FUNCTION_BLOCK FB_NovRamToFileRingBuffer
VAR_INPUT
	udiNovRamIndex:UDINT;
	dataType:DINT;
END_VAR
VAR_OUTPUT
	//readData:ARRAY [0..GVL.arrArrayLength[E_DB_StructureType.AlarmHistory]-1] OF ST_AlarmInfo_DB_save;
END_VAR
VAR
END_VAR
VAR_IN_OUT
	NovRamData:ST_NovRam;
END_VAR

IF dataType = E_DB_StructureType.AlarmHistory THEN
	M_AlarmHistory(udiNovRamIndex:=udiNovRamIndex);
ELSIF dataType = E_DB_StructureType.ProductionHistory THEN
	M_ProductionHistory(udiNovRamIndex:=udiNovRamIndex);
ELSIF dataType = E_DB_StructureType.ProductionReport THEN
	M_ProductionReport(udiNovRamIndex:=udiNovRamIndex);
ELSIF dataType = E_DB_StructureType.ProductionSummary THEN
	M_ProductionSummary(udiNovRamIndex:=udiNovRamIndex);
ELSIF dataType = E_DB_StructureType.SoDuration THEN
	M_SoDuration(udiNovRamIndex:=udiNovRamIndex);
ELSIF dataType = E_DB_StructureType.StopCount THEN
	M_StopCount(udiNovRamIndex:=udiNovRamIndex);
ELSIF dataType = E_DB_StructureType.RegularCheckResults THEN
	M_RegularCheckResults(udiNovRamIndex:=udiNovRamIndex);
END_IF

METHOD M_AlarmHistory : BOOL
VAR_INPUT
	udiNovRamIndex:UDINT;
END_VAR
VAR_OUTPUT
	
END_VAR
VAR_INST
	WriteData:ARRAY[0..GVL.arrArrayLength[E_DB_StructureType.AlarmHistory]-1] OF ST_AlarmInfo_DB_save;//small
	iStep:INT;
	i:UDINT;
	fbFileRingBuffer: FB_FileRingBuffer := ( sNetId     := '',
                                             sPathName  := '',
                                             ePath      := PATH_GENERIC,
                                             nID        := 1,
                                             cbBuffer   := gvl.arrFileRingBufferSize[E_DB_StructureType.AlarmHistory], //5MB(5*10^6Bytes)
                                             bOverwrite := FALSE,
                                             pWriteBuff := 0,
                                             cbWriteLen := 0,
                                             pReadBuff  := 0,
                                             cbReadLen  := 0,
                                             tTimeout   := T#1S );
	bBusy:BOOL;
	bError:BOOL;
	nErrID:UDINT;
	stHeader:ST_FileRBufferHead;
    loadData  : ARRAY[0..511] OF BYTE :=[512(0)];
    cbLoad    : UDINT;
	
	fileName:STRING(255);
	tempFileIndex:UDINT;
	eStrIndex:DINT;
	
	//1217
	TransTrig:TON;
END_VAR
//Config	
eStrIndex:=E_DB_StructureType.AlarmHistory;

fbFileRingBuffer(sPathName:=fileName
				,bBusy=>bBusy,bError=>bError,nErrID=>nErrID
				,cbReturn=>cbLoad,stHeader=>stHeader);
//1217				
TransTrig(PT:=T#10S);//10s upload one time

CASE iStep OF
	0://NovRam full detect / file full detect
		
		tempFileIndex:=NovRamData.arrFileRingBuffer_Status[eStrIndex].nowFileIndex[udiNovRamIndex];
		
		//1217
		IF NovRamData.arrNovRam_Status[eStrIndex].RowDataLocked[udiNovRamIndex] = FALSE//not full and 
		AND NovRamData.arrNovRam_Status[eStrIndex].writenIndex > 0 THEN//has been writen
			
			TransTrig(IN:=TRUE);
			
			IF TransTrig.Q //timeout
			AND NovRamData.arrFileRingBuffer_Status[eStrIndex].bFileFull[udiNovRamIndex][tempFileIndex] = FALSE THEN//File can write
				TransTrig(IN:=FALSE);
				
				//Set Row Lock
				NovRamData.arrNovRam_Status[eStrIndex].RowDataLocked[udiNovRamIndex]:=TRUE;
				
				//save writen count
				NovRamData.arrNovRam_Status[eStrIndex].writenCount := NovRamData.arrNovRam_Status[eStrIndex].writenIndex;
				
				//Reset Row and writenIndex
				NovRamData.arrNovRam_Status[eStrIndex].nowRowIndex:=(udiNovRamIndex+1)MOD GVL.NovRamBufferRatio;
				NovRamData.arrNovRam_Status[eStrIndex].writenIndex:=0;
		
				fileName:=M_GetFileName(structureType:=eStrIndex
										,udiNovRam_BufferIndex:=udiNovRamIndex
										,udiFile_Index:=NovRamData.arrFileRingBuffer_Status[eStrIndex].nowFileIndex[udiNovRamIndex]);
										
				iStep:=1;
			END_IF
			
		ELSE
			IF NovRamData.arrNovRam_Status[eStrIndex].RowDataLocked[udiNovRamIndex] //NovRam full = should work
			AND NovRamData.arrFileRingBuffer_Status[eStrIndex].bFileFull[udiNovRamIndex][tempFileIndex] = FALSE//File can write
			THEN
				//
				fileName:=M_GetFileName(structureType:=eStrIndex
										,udiNovRam_BufferIndex:=udiNovRamIndex
										,udiFile_Index:=NovRamData.arrFileRingBuffer_Status[eStrIndex].nowFileIndex[udiNovRamIndex]);
										
				iStep:=1;
			END_IF
		END_IF
		
		

	1://Open File
		
		fbFileRingBuffer.A_Open();
		
		iStep:=2;
		
	2://Wait Done/Add Data
		IF fbFileRingBuffer.bBusy=FALSE AND NOT fbFileRingBuffer.bError THEN
			
			//1217
			//FOR i:=0 TO GVL.arrArrayLength[E_DB_StructureType.AlarmHistory]-1 DO 
			FOR i:=0 TO NovRamData.arrNovRam_Status[eStrIndex].writenCount-1 DO
				WriteData[i] := NovRamData.AlarmHistory[udiNovRamIndex][i];
			END_FOR
			
			//1217
			//Add
			//fbFileRingBuffer.A_AddTail( pWriteBuff := ADR(WriteData), cbWriteLen := SIZEOF(WriteData),
			//		pReadBuff := 0, cbReadLen:=0 );
			fbFileRingBuffer.A_AddTail( pWriteBuff := ADR(WriteData), cbWriteLen := NovRamData.arrNovRam_Status[eStrIndex].writenCount * SIZEOF(ST_AlarmInfo_DB_save),
					pReadBuff := 0, cbReadLen:=0 );
					
			iStep:=3;
			
		END_IF
	3://Wait Done / Close file /(Check if file Full)
		IF fbFileRingBuffer.bBusy=FALSE THEN
						
			//Check if file full
			IF NOT fbFileRingBuffer.bError THEN
				iStep:=4;
			ELSIF fbFileRingBuffer.bError = TRUE AND nErrID=32768 THEN//full
				iStep:=11;
			END_IF
			
			//close file
			fbFileRingBuffer.A_Close();
			
		END_IF
	4://Wait Done(file still has space)
		IF fbFileRingBuffer.bBusy=FALSE AND NOT fbFileRingBuffer.bError THEN
			
			NovRamData.arrNovRam_Status[eStrIndex].RowDataLocked[udiNovRamIndex]:=FALSE;
			
			iStep:=0;
		END_IF
	11://Wait Done(file full)
		IF fbFileRingBuffer.bBusy=FALSE AND NOT fbFileRingBuffer.bError THEN
			
			//Lock now file
			//NovRamData.arrFileRingBuffer_Status.bFileFull[(gvl.FileRingBufferRatio * udiNovRamIndex) + NovRamData.arrFileRingBuffer_Status.nowFileIndex[udiNovRamIndex]]:=TRUE;
			tempFileIndex:=NovRamData.arrFileRingBuffer_Status[eStrIndex].nowFileIndex[udiNovRamIndex];
			NovRamData.arrFileRingBuffer_Status[eStrIndex].bFileFull[udiNovRamIndex][tempFileIndex]:=TRUE;
			
			//Move to next FileIndex
			NovRamData.arrFileRingBuffer_Status[eStrIndex].nowFileIndex[udiNovRamIndex]:=((NovRamData.arrFileRingBuffer_Status[eStrIndex].nowFileIndex[udiNovRamIndex]+1) MOD GVL.FileRingBufferRatio);
			
			iStep:=0;
			
		END_IF
END_CASE
END_METHOD

METHOD M_GetFileName : STRING(255)
VAR_INPUT
	structureType:DINT;
	udiNovRam_BufferIndex:UDINT;
	udiFile_Index:UDINT;
END_VAR
VAR
	tempString:STRING(255);
	tempString2:STRING(255);
	tempFileNo:UDINT;
END_VAR
IF structureType=E_DB_StructureType.AlarmHistory THEN
	tempString:=CONCAT(gvl.arrfileFolder[structureType],'AlarmHistory');
ELSIF structureType=E_DB_StructureType.ProductionHistory THEN
	tempString:=CONCAT(gvl.arrfileFolder[structureType],'ProductionHistory');
ELSIF structureType=E_DB_StructureType.ProductionReport THEN
	tempString:=CONCAT(gvl.arrfileFolder[structureType],'ProductionReport');
ELSIF structureType=E_DB_StructureType.ProductionSummary THEN
	tempString:=CONCAT(gvl.arrfileFolder[structureType],'ProductionSummary');
ELSIF structureType=E_DB_StructureType.SoDuration THEN
	tempString:=CONCAT(gvl.arrfileFolder[structureType],'SoDuration');
ELSIF structureType=E_DB_StructureType.StopCount THEN
	tempString:=CONCAT(gvl.arrfileFolder[structureType],'StopCount');
ELSIF structureType=E_DB_StructureType.RegularCheckResults THEN
	tempString:=CONCAT(gvl.arrfileFolder[structureType],'RegularCheckResults');
END_IF

tempFileNo:=(udiNovRam_BufferIndex) * GVL.FileRingBufferRatio + (udiFile_Index + 1);
tempString2:=CONCAT(tempString,UDINT_TO_STRING(tempFileNo));
M_GetFileName:=CONCAT(tempString2,'.dat');
END_METHOD

METHOD M_ProductionHistory : BOOL
VAR_INPUT
	udiNovRamIndex:UDINT;
END_VAR
VAR_INST
	WriteData:ARRAY[0..GVL.arrArrayLength[E_DB_StructureType.ProductionHistory]-1] OF ST_PHI_GroupData_DB;//small
	iStep:INT;
	i:UDINT;
	fbFileRingBuffer: FB_FileRingBuffer := ( sNetId     := '',
                                             sPathName  := '',
                                             ePath      := PATH_GENERIC,
                                             nID        := 1,
                                             cbBuffer   := gvl.arrFileRingBufferSize[E_DB_StructureType.ProductionHistory], //5MB(5*10^6Bytes)
                                             bOverwrite := FALSE,
                                             pWriteBuff := 0,
                                             cbWriteLen := 0,
                                             pReadBuff  := 0,
                                             cbReadLen  := 0,
                                             tTimeout   := T#1S );
	bBusy:BOOL;
	bError:BOOL;
	nErrID:UDINT;
	stHeader:ST_FileRBufferHead;
    loadData  : ARRAY[0..511] OF BYTE :=[512(0)];
    cbLoad    : UDINT;
	
	fileName:STRING(255);
	tempFileIndex:UDINT;
	eStrIndex:DINT;
END_VAR
//Config
eStrIndex:=E_DB_StructureType.ProductionHistory;

fbFileRingBuffer(sPathName:=fileName
				,bBusy=>bBusy,bError=>bError,nErrID=>nErrID
				,cbReturn=>cbLoad,stHeader=>stHeader);

CASE iStep OF
	0://NovRam full detect / file full detect
		
		tempFileIndex:=NovRamData.arrFileRingBuffer_Status[eStrIndex].nowFileIndex[udiNovRamIndex];
		
		IF NovRamData.arrNovRam_Status[eStrIndex].RowDataLocked[udiNovRamIndex] //NovRam full = should work
		AND NovRamData.arrFileRingBuffer_Status[eStrIndex].bFileFull[udiNovRamIndex][tempFileIndex] = FALSE//File can write
		THEN
			//
			fileName:=M_GetFileName(structureType:=eStrIndex
									,udiNovRam_BufferIndex:=udiNovRamIndex
									,udiFile_Index:=NovRamData.arrFileRingBuffer_Status[eStrIndex].nowFileIndex[udiNovRamIndex]);
									
			iStep:=1;
		END_IF

	1://Open File
		
		fbFileRingBuffer.A_Open();
		
		iStep:=2;
		
	2://Wait Done/Add Data
		IF fbFileRingBuffer.bBusy=FALSE AND NOT fbFileRingBuffer.bError THEN
			
			FOR i:=0 TO GVL.arrArrayLength[E_DB_StructureType.ProductionHistory]-1 DO 
				WriteData[i] := NovRamData.ProductionHistory[udiNovRamIndex][i];
			END_FOR
			
			//Add
			fbFileRingBuffer.A_AddTail( pWriteBuff := ADR(WriteData), cbWriteLen := SIZEOF(WriteData),
					pReadBuff := 0, cbReadLen:=0 );
			
			iStep:=3;
			
		END_IF
	3://Wait Done / Close file /(Check if file Full)
		IF fbFileRingBuffer.bBusy=FALSE THEN
						
			//Check if file full
			IF NOT fbFileRingBuffer.bError THEN
				iStep:=4;
			ELSIF fbFileRingBuffer.bError = TRUE AND nErrID=32768 THEN//full
				iStep:=11;
			END_IF
			
			//close file
			fbFileRingBuffer.A_Close();
			
		END_IF
	4://Wait Done(file still has space)
		IF fbFileRingBuffer.bBusy=FALSE AND NOT fbFileRingBuffer.bError THEN
			
			NovRamData.arrNovRam_Status[eStrIndex].RowDataLocked[udiNovRamIndex]:=FALSE;
			
			iStep:=0;
		END_IF
	11://Wait Done(file full)
		IF fbFileRingBuffer.bBusy=FALSE AND NOT fbFileRingBuffer.bError THEN
			
			//Lock now file
			//NovRamData.FileRingBuffer_Status.bFileFull[(gvl.FileRingBufferRatio * udiNovRamIndex) + NovRamData.FileRingBuffer_Status.nowFileIndex[udiNovRamIndex]]:=TRUE;
			tempFileIndex:=NovRamData.arrFileRingBuffer_Status[eStrIndex].nowFileIndex[udiNovRamIndex];
			NovRamData.arrFileRingBuffer_Status[eStrIndex].bFileFull[udiNovRamIndex][tempFileIndex]:=TRUE;
			
			//Move to next FileIndex
			NovRamData.arrFileRingBuffer_Status[eStrIndex].nowFileIndex[udiNovRamIndex]:=((NovRamData.arrFileRingBuffer_Status[eStrIndex].nowFileIndex[udiNovRamIndex]+1) MOD GVL.FileRingBufferRatio);
			
			iStep:=0;
			
		END_IF
END_CASE
END_METHOD

METHOD M_ProductionReport : BOOL
VAR_INPUT
	udiNovRamIndex:UDINT;
END_VAR
VAR_INST
	WriteData:ARRAY[0..GVL.arrArrayLength[E_DB_StructureType.ProductionReport]-1] OF ST_OEE_ProductionReport;//small
	iStep:INT;
	i:UDINT;
	fbFileRingBuffer: FB_FileRingBuffer := ( sNetId     := '',
                                             sPathName  := '',
                                             ePath      := PATH_GENERIC,
                                             nID        := 1,
                                             cbBuffer   := gvl.arrFileRingBufferSize[E_DB_StructureType.ProductionReport], //5MB(5*10^6Bytes)
                                             bOverwrite := FALSE,
                                             pWriteBuff := 0,
                                             cbWriteLen := 0,
                                             pReadBuff  := 0,
                                             cbReadLen  := 0,
                                             tTimeout   := T#1S );
	bBusy:BOOL;
	bError:BOOL;
	nErrID:UDINT;
	stHeader:ST_FileRBufferHead;
    loadData  : ARRAY[0..511] OF BYTE :=[512(0)];
    cbLoad    : UDINT;
	
	fileName:STRING(255);
	tempFileIndex:UDINT;
	eStrIndex:DINT;
END_VAR
//Config
eStrIndex:=E_DB_StructureType.ProductionReport;

fbFileRingBuffer(sPathName:=fileName
				,bBusy=>bBusy,bError=>bError,nErrID=>nErrID
				,cbReturn=>cbLoad,stHeader=>stHeader);

CASE iStep OF
	0://NovRam full detect / file full detect
		
		tempFileIndex:=NovRamData.arrFileRingBuffer_Status[eStrIndex].nowFileIndex[udiNovRamIndex];
		
		IF NovRamData.arrNovRam_Status[eStrIndex].RowDataLocked[udiNovRamIndex] //NovRam full = should work
		AND NovRamData.arrFileRingBuffer_Status[eStrIndex].bFileFull[udiNovRamIndex][tempFileIndex] = FALSE//File can write
		THEN
			//
			fileName:=M_GetFileName(structureType:=eStrIndex
									,udiNovRam_BufferIndex:=udiNovRamIndex
									,udiFile_Index:=NovRamData.arrFileRingBuffer_Status[eStrIndex].nowFileIndex[udiNovRamIndex]);
									
			iStep:=1;
		END_IF

	1://Open File
		
		fbFileRingBuffer.A_Open();
		
		iStep:=2;
		
	2://Wait Done/Add Data
		IF fbFileRingBuffer.bBusy=FALSE AND NOT fbFileRingBuffer.bError THEN
			
			FOR i:=0 TO GVL.arrArrayLength[E_DB_StructureType.ProductionReport]-1 DO 
				WriteData[i] := NovRamData.ProductionReport[udiNovRamIndex][i];
			END_FOR
			
			//Add
			fbFileRingBuffer.A_AddTail( pWriteBuff := ADR(WriteData), cbWriteLen := SIZEOF(WriteData),
					pReadBuff := 0, cbReadLen:=0 );
			
			iStep:=3;
			
		END_IF
	3://Wait Done / Close file /(Check if file Full)
		IF fbFileRingBuffer.bBusy=FALSE THEN
						
			//Check if file full
			IF NOT fbFileRingBuffer.bError THEN
				iStep:=4;
			ELSIF fbFileRingBuffer.bError = TRUE AND nErrID=32768 THEN//full
				iStep:=11;
			END_IF
			
			//close file
			fbFileRingBuffer.A_Close();
			
		END_IF
	4://Wait Done(file still has space)
		IF fbFileRingBuffer.bBusy=FALSE AND NOT fbFileRingBuffer.bError THEN
			
			NovRamData.arrNovRam_Status[eStrIndex].RowDataLocked[udiNovRamIndex]:=FALSE;
			
			iStep:=0;
		END_IF
	11://Wait Done(file full)
		IF fbFileRingBuffer.bBusy=FALSE AND NOT fbFileRingBuffer.bError THEN
			
			//Lock now file
			//NovRamData.FileRingBuffer_Status.bFileFull[(gvl.FileRingBufferRatio * udiNovRamIndex) + NovRamData.FileRingBuffer_Status.nowFileIndex[udiNovRamIndex]]:=TRUE;
			tempFileIndex:=NovRamData.arrFileRingBuffer_Status[eStrIndex].nowFileIndex[udiNovRamIndex];
			NovRamData.arrFileRingBuffer_Status[eStrIndex].bFileFull[udiNovRamIndex][tempFileIndex]:=TRUE;
			
			//Move to next FileIndex
			NovRamData.arrFileRingBuffer_Status[eStrIndex].nowFileIndex[udiNovRamIndex]:=((NovRamData.arrFileRingBuffer_Status[eStrIndex].nowFileIndex[udiNovRamIndex]+1) MOD GVL.FileRingBufferRatio);
			
			iStep:=0;
			
		END_IF
END_CASE
END_METHOD

METHOD M_ProductionSummary : BOOL
VAR_INPUT
	udiNovRamIndex:UDINT;
END_VAR
VAR_INST
	WriteData:ARRAY[0..GVL.arrArrayLength[E_DB_StructureType.ProductionSummary]-1] OF ST_OEE_ProductionSummary;//small
	iStep:INT;
	i:UDINT;
	fbFileRingBuffer: FB_FileRingBuffer := ( sNetId     := '',
                                             sPathName  := '',
                                             ePath      := PATH_GENERIC,
                                             nID        := 1,
                                             cbBuffer   := gvl.arrFileRingBufferSize[E_DB_StructureType.ProductionSummary], //5MB(5*10^6Bytes)
                                             bOverwrite := FALSE,
                                             pWriteBuff := 0,
                                             cbWriteLen := 0,
                                             pReadBuff  := 0,
                                             cbReadLen  := 0,
                                             tTimeout   := T#1S );
	bBusy:BOOL;
	bError:BOOL;
	nErrID:UDINT;
	stHeader:ST_FileRBufferHead;
    loadData  : ARRAY[0..511] OF BYTE :=[512(0)];
    cbLoad    : UDINT;
	
	fileName:STRING(255);
	tempFileIndex:UDINT;
	eStrIndex:DINT;
END_VAR
//Config
eStrIndex:=E_DB_StructureType.ProductionSummary;

fbFileRingBuffer(sPathName:=fileName
				,bBusy=>bBusy,bError=>bError,nErrID=>nErrID
				,cbReturn=>cbLoad,stHeader=>stHeader);

CASE iStep OF
	0://NovRam full detect / file full detect
		
		tempFileIndex:=NovRamData.arrFileRingBuffer_Status[eStrIndex].nowFileIndex[udiNovRamIndex];
		
		IF NovRamData.arrNovRam_Status[eStrIndex].RowDataLocked[udiNovRamIndex] //NovRam full = should work
		AND NovRamData.arrFileRingBuffer_Status[eStrIndex].bFileFull[udiNovRamIndex][tempFileIndex] = FALSE//File can write
		THEN
			//
			fileName:=M_GetFileName(structureType:=eStrIndex
									,udiNovRam_BufferIndex:=udiNovRamIndex
									,udiFile_Index:=NovRamData.arrFileRingBuffer_Status[eStrIndex].nowFileIndex[udiNovRamIndex]);
									
			iStep:=1;
		END_IF

	1://Open File
		
		fbFileRingBuffer.A_Open();
		
		iStep:=2;
		
	2://Wait Done/Add Data
		IF fbFileRingBuffer.bBusy=FALSE AND NOT fbFileRingBuffer.bError THEN
			
			FOR i:=0 TO GVL.arrArrayLength[E_DB_StructureType.ProductionSummary]-1 DO 
				WriteData[i] := NovRamData.ProductionSummary[udiNovRamIndex][i];
			END_FOR
			
			//Add
			fbFileRingBuffer.A_AddTail( pWriteBuff := ADR(WriteData), cbWriteLen := SIZEOF(WriteData),
					pReadBuff := 0, cbReadLen:=0 );
			
			iStep:=3;
			
		END_IF
	3://Wait Done / Close file /(Check if file Full)
		IF fbFileRingBuffer.bBusy=FALSE THEN
						
			//Check if file full
			IF NOT fbFileRingBuffer.bError THEN
				iStep:=4;
			ELSIF fbFileRingBuffer.bError = TRUE AND nErrID=32768 THEN//full
				iStep:=11;
			END_IF
			
			//close file
			fbFileRingBuffer.A_Close();
			
		END_IF
	4://Wait Done(file still has space)
		IF fbFileRingBuffer.bBusy=FALSE AND NOT fbFileRingBuffer.bError THEN
			
			NovRamData.arrNovRam_Status[eStrIndex].RowDataLocked[udiNovRamIndex]:=FALSE;
			
			iStep:=0;
		END_IF
	11://Wait Done(file full)
		IF fbFileRingBuffer.bBusy=FALSE AND NOT fbFileRingBuffer.bError THEN
			
			//Lock now file
			//NovRamData.FileRingBuffer_Status.bFileFull[(gvl.FileRingBufferRatio * udiNovRamIndex) + NovRamData.FileRingBuffer_Status.nowFileIndex[udiNovRamIndex]]:=TRUE;
			tempFileIndex:=NovRamData.arrFileRingBuffer_Status[eStrIndex].nowFileIndex[udiNovRamIndex];
			NovRamData.arrFileRingBuffer_Status[eStrIndex].bFileFull[udiNovRamIndex][tempFileIndex]:=TRUE;
			
			//Move to next FileIndex
			NovRamData.arrFileRingBuffer_Status[eStrIndex].nowFileIndex[udiNovRamIndex]:=((NovRamData.arrFileRingBuffer_Status[eStrIndex].nowFileIndex[udiNovRamIndex]+1) MOD GVL.FileRingBufferRatio);
			
			iStep:=0;
			
		END_IF
END_CASE
END_METHOD

METHOD M_RegularCheckResults : BOOL
VAR_INPUT
	udiNovRamIndex:UDINT;
END_VAR
VAR_INST
	WriteData:ARRAY[0..GVL.arrArrayLength[E_DB_StructureType.RegularCheckResults]-1] OF ST_RegularCheck_Results;//small
	iStep:INT;
	i:UDINT;
	fbFileRingBuffer: FB_FileRingBuffer := ( sNetId     := '',
                                             sPathName  := '',
                                             ePath      := PATH_GENERIC,
                                             nID        := 1,
                                             cbBuffer   := gvl.arrFileRingBufferSize[E_DB_StructureType.RegularCheckResults], //5MB(5*10^6Bytes)
                                             bOverwrite := FALSE,
                                             pWriteBuff := 0,
                                             cbWriteLen := 0,
                                             pReadBuff  := 0,
                                             cbReadLen  := 0,
                                             tTimeout   := T#1S );
	bBusy:BOOL;
	bError:BOOL;
	nErrID:UDINT;
	stHeader:ST_FileRBufferHead;
    loadData  : ARRAY[0..511] OF BYTE :=[512(0)];
    cbLoad    : UDINT;
	
	fileName:STRING(255);
	tempFileIndex:UDINT;
	eStrIndex:DINT;
END_VAR
//Config
eStrIndex:=E_DB_StructureType.RegularCheckResults;

fbFileRingBuffer(sPathName:=fileName
				,bBusy=>bBusy,bError=>bError,nErrID=>nErrID
				,cbReturn=>cbLoad,stHeader=>stHeader);

CASE iStep OF
	0://NovRam full detect / file full detect
		
		tempFileIndex:=NovRamData.arrFileRingBuffer_Status[eStrIndex].nowFileIndex[udiNovRamIndex];
		
		IF NovRamData.arrNovRam_Status[eStrIndex].RowDataLocked[udiNovRamIndex] //NovRam full = should work
		AND NovRamData.arrFileRingBuffer_Status[eStrIndex].bFileFull[udiNovRamIndex][tempFileIndex] = FALSE//File can write
		THEN
			//
			fileName:=M_GetFileName(structureType:=eStrIndex
									,udiNovRam_BufferIndex:=udiNovRamIndex
									,udiFile_Index:=NovRamData.arrFileRingBuffer_Status[eStrIndex].nowFileIndex[udiNovRamIndex]);
									
			iStep:=1;
		END_IF

	1://Open File
		
		fbFileRingBuffer.A_Open();
		
		iStep:=2;
		
	2://Wait Done/Add Data
		IF fbFileRingBuffer.bBusy=FALSE AND NOT fbFileRingBuffer.bError THEN
			
			FOR i:=0 TO GVL.arrArrayLength[E_DB_StructureType.RegularCheckResults]-1 DO 
				WriteData[i] := NovRamData.RegularCheckResults[udiNovRamIndex][i];
			END_FOR
			
			//Add
			fbFileRingBuffer.A_AddTail( pWriteBuff := ADR(WriteData), cbWriteLen := SIZEOF(WriteData),
					pReadBuff := 0, cbReadLen:=0 );
			
			iStep:=3;
			
		END_IF
	3://Wait Done / Close file /(Check if file Full)
		IF fbFileRingBuffer.bBusy=FALSE THEN
						
			//Check if file full
			IF NOT fbFileRingBuffer.bError THEN
				iStep:=4;
			ELSIF fbFileRingBuffer.bError = TRUE AND nErrID=32768 THEN//full
				iStep:=11;
			END_IF
			
			//close file
			fbFileRingBuffer.A_Close();
			
		END_IF
	4://Wait Done(file still has space)
		IF fbFileRingBuffer.bBusy=FALSE AND NOT fbFileRingBuffer.bError THEN
			
			NovRamData.arrNovRam_Status[eStrIndex].RowDataLocked[udiNovRamIndex]:=FALSE;
			
			iStep:=0;
		END_IF
	11://Wait Done(file full)
		IF fbFileRingBuffer.bBusy=FALSE AND NOT fbFileRingBuffer.bError THEN
			
			//Lock now file
			//NovRamData.FileRingBuffer_Status.bFileFull[(gvl.FileRingBufferRatio * udiNovRamIndex) + NovRamData.FileRingBuffer_Status.nowFileIndex[udiNovRamIndex]]:=TRUE;
			tempFileIndex:=NovRamData.arrFileRingBuffer_Status[eStrIndex].nowFileIndex[udiNovRamIndex];
			NovRamData.arrFileRingBuffer_Status[eStrIndex].bFileFull[udiNovRamIndex][tempFileIndex]:=TRUE;
			
			//Move to next FileIndex
			NovRamData.arrFileRingBuffer_Status[eStrIndex].nowFileIndex[udiNovRamIndex]:=((NovRamData.arrFileRingBuffer_Status[eStrIndex].nowFileIndex[udiNovRamIndex]+1) MOD GVL.FileRingBufferRatio);
			
			iStep:=0;
			
		END_IF
END_CASE
END_METHOD

METHOD M_SoDuration : BOOL
VAR_INPUT
	udiNovRamIndex:UDINT;
END_VAR
VAR_INST
	WriteData:ARRAY[0..GVL.arrArrayLength[E_DB_StructureType.SoDuration]-1] OF ST_SoDuration;//small
	iStep:INT;
	i:UDINT;
	fbFileRingBuffer: FB_FileRingBuffer := ( sNetId     := '',
                                             sPathName  := '',
                                             ePath      := PATH_GENERIC,
                                             nID        := 1,
                                             cbBuffer   := gvl.arrFileRingBufferSize[E_DB_StructureType.SoDuration], //5MB(5*10^6Bytes)
                                             bOverwrite := FALSE,
                                             pWriteBuff := 0,
                                             cbWriteLen := 0,
                                             pReadBuff  := 0,
                                             cbReadLen  := 0,
                                             tTimeout   := T#1S );
	bBusy:BOOL;
	bError:BOOL;
	nErrID:UDINT;
	stHeader:ST_FileRBufferHead;
    loadData  : ARRAY[0..511] OF BYTE :=[512(0)];
    cbLoad    : UDINT;
	
	fileName:STRING(255);
	tempFileIndex:UDINT;
	eStrIndex:DINT;
END_VAR
//Config
eStrIndex:=E_DB_StructureType.SoDuration;

fbFileRingBuffer(sPathName:=fileName
				,bBusy=>bBusy,bError=>bError,nErrID=>nErrID
				,cbReturn=>cbLoad,stHeader=>stHeader);

CASE iStep OF
	0://NovRam full detect / file full detect
		
		tempFileIndex:=NovRamData.arrFileRingBuffer_Status[eStrIndex].nowFileIndex[udiNovRamIndex];
		
		IF NovRamData.arrNovRam_Status[eStrIndex].RowDataLocked[udiNovRamIndex] //NovRam full = should work
		AND NovRamData.arrFileRingBuffer_Status[eStrIndex].bFileFull[udiNovRamIndex][tempFileIndex] = FALSE//File can write
		THEN
			//
			fileName:=M_GetFileName(structureType:=eStrIndex
									,udiNovRam_BufferIndex:=udiNovRamIndex
									,udiFile_Index:=NovRamData.arrFileRingBuffer_Status[eStrIndex].nowFileIndex[udiNovRamIndex]);
									
			iStep:=1;
		END_IF

	1://Open File
		
		fbFileRingBuffer.A_Open();
		
		iStep:=2;
		
	2://Wait Done/Add Data
		IF fbFileRingBuffer.bBusy=FALSE AND NOT fbFileRingBuffer.bError THEN
			
			FOR i:=0 TO GVL.arrArrayLength[E_DB_StructureType.SoDuration]-1 DO 
				WriteData[i] := NovRamData.SoDuration[udiNovRamIndex][i];
			END_FOR
			
			//Add
			fbFileRingBuffer.A_AddTail( pWriteBuff := ADR(WriteData), cbWriteLen := SIZEOF(WriteData),
					pReadBuff := 0, cbReadLen:=0 );
			
			iStep:=3;
			
		END_IF
	3://Wait Done / Close file /(Check if file Full)
		IF fbFileRingBuffer.bBusy=FALSE THEN
						
			//Check if file full
			IF NOT fbFileRingBuffer.bError THEN
				iStep:=4;
			ELSIF fbFileRingBuffer.bError = TRUE AND nErrID=32768 THEN//full
				iStep:=11;
			END_IF
			
			//close file
			fbFileRingBuffer.A_Close();
			
		END_IF
	4://Wait Done(file still has space)
		IF fbFileRingBuffer.bBusy=FALSE AND NOT fbFileRingBuffer.bError THEN
			
			NovRamData.arrNovRam_Status[eStrIndex].RowDataLocked[udiNovRamIndex]:=FALSE;
			
			iStep:=0;
		END_IF
	11://Wait Done(file full)
		IF fbFileRingBuffer.bBusy=FALSE AND NOT fbFileRingBuffer.bError THEN
			
			//Lock now file
			//NovRamData.FileRingBuffer_Status.bFileFull[(gvl.FileRingBufferRatio * udiNovRamIndex) + NovRamData.FileRingBuffer_Status.nowFileIndex[udiNovRamIndex]]:=TRUE;
			tempFileIndex:=NovRamData.arrFileRingBuffer_Status[eStrIndex].nowFileIndex[udiNovRamIndex];
			NovRamData.arrFileRingBuffer_Status[eStrIndex].bFileFull[udiNovRamIndex][tempFileIndex]:=TRUE;
			
			//Move to next FileIndex
			NovRamData.arrFileRingBuffer_Status[eStrIndex].nowFileIndex[udiNovRamIndex]:=((NovRamData.arrFileRingBuffer_Status[eStrIndex].nowFileIndex[udiNovRamIndex]+1) MOD GVL.FileRingBufferRatio);
			
			iStep:=0;
			
		END_IF
END_CASE
END_METHOD

METHOD M_StopCount : BOOL
VAR_INPUT
	udiNovRamIndex:UDINT;
END_VAR
VAR_INST
	WriteData:ARRAY[0..GVL.arrArrayLength[E_DB_StructureType.StopCount]-1] OF ST_StopCount;//small
	iStep:INT;
	i:UDINT;
	fbFileRingBuffer: FB_FileRingBuffer := ( sNetId     := '',
                                             sPathName  := '',
                                             ePath      := PATH_GENERIC,
                                             nID        := 1,
                                             cbBuffer   := gvl.arrFileRingBufferSize[E_DB_StructureType.StopCount], //5MB(5*10^6Bytes)
                                             bOverwrite := FALSE,
                                             pWriteBuff := 0,
                                             cbWriteLen := 0,
                                             pReadBuff  := 0,
                                             cbReadLen  := 0,
                                             tTimeout   := T#1S );
	bBusy:BOOL;
	bError:BOOL;
	nErrID:UDINT;
	stHeader:ST_FileRBufferHead;
    loadData  : ARRAY[0..511] OF BYTE :=[512(0)];
    cbLoad    : UDINT;
	
	fileName:STRING(255);
	tempFileIndex:UDINT;
	eStrIndex:DINT;
END_VAR
//Config
eStrIndex:=E_DB_StructureType.StopCount;

fbFileRingBuffer(sPathName:=fileName
				,bBusy=>bBusy,bError=>bError,nErrID=>nErrID
				,cbReturn=>cbLoad,stHeader=>stHeader);

CASE iStep OF
	0://NovRam full detect / file full detect
		
		tempFileIndex:=NovRamData.arrFileRingBuffer_Status[eStrIndex].nowFileIndex[udiNovRamIndex];
		
		IF NovRamData.arrNovRam_Status[eStrIndex].RowDataLocked[udiNovRamIndex] //NovRam full = should work
		AND NovRamData.arrFileRingBuffer_Status[eStrIndex].bFileFull[udiNovRamIndex][tempFileIndex] = FALSE//File can write
		THEN
			//
			fileName:=M_GetFileName(structureType:=eStrIndex
									,udiNovRam_BufferIndex:=udiNovRamIndex
									,udiFile_Index:=NovRamData.arrFileRingBuffer_Status[eStrIndex].nowFileIndex[udiNovRamIndex]);
									
			iStep:=1;
		END_IF

	1://Open File
		
		fbFileRingBuffer.A_Open();
		
		iStep:=2;
		
	2://Wait Done/Add Data
		IF fbFileRingBuffer.bBusy=FALSE AND NOT fbFileRingBuffer.bError THEN
			
			FOR i:=0 TO GVL.arrArrayLength[E_DB_StructureType.StopCount]-1 DO 
				WriteData[i] := NovRamData.StopCount[udiNovRamIndex][i];
			END_FOR
			
			//Add
			fbFileRingBuffer.A_AddTail( pWriteBuff := ADR(WriteData), cbWriteLen := SIZEOF(WriteData),
					pReadBuff := 0, cbReadLen:=0 );
			
			iStep:=3;
			
		END_IF
	3://Wait Done / Close file /(Check if file Full)
		IF fbFileRingBuffer.bBusy=FALSE THEN
						
			//Check if file full
			IF NOT fbFileRingBuffer.bError THEN
				iStep:=4;
			ELSIF fbFileRingBuffer.bError = TRUE AND nErrID=32768 THEN//full
				iStep:=11;
			END_IF
			
			//close file
			fbFileRingBuffer.A_Close();
			
		END_IF
	4://Wait Done(file still has space)
		IF fbFileRingBuffer.bBusy=FALSE AND NOT fbFileRingBuffer.bError THEN
			
			NovRamData.arrNovRam_Status[eStrIndex].RowDataLocked[udiNovRamIndex]:=FALSE;
			
			iStep:=0;
		END_IF
	11://Wait Done(file full)
		IF fbFileRingBuffer.bBusy=FALSE AND NOT fbFileRingBuffer.bError THEN
			
			//Lock now file
			//NovRamData.FileRingBuffer_Status.bFileFull[(gvl.FileRingBufferRatio * udiNovRamIndex) + NovRamData.FileRingBuffer_Status.nowFileIndex[udiNovRamIndex]]:=TRUE;
			tempFileIndex:=NovRamData.arrFileRingBuffer_Status[eStrIndex].nowFileIndex[udiNovRamIndex];
			NovRamData.arrFileRingBuffer_Status[eStrIndex].bFileFull[udiNovRamIndex][tempFileIndex]:=TRUE;
			
			//Move to next FileIndex
			NovRamData.arrFileRingBuffer_Status[eStrIndex].nowFileIndex[udiNovRamIndex]:=((NovRamData.arrFileRingBuffer_Status[eStrIndex].nowFileIndex[udiNovRamIndex]+1) MOD GVL.FileRingBufferRatio);
			
			iStep:=0;
			
		END_IF
END_CASE
END_METHOD

END_FUNCTION_BLOCK

(* stored: Version 1.1.0.1, ProductVersion 3.1.4024.11
   POU FB_NovRamToFileRingBuffer: Id {c9bcde8f-ded9-4a08-b333-ef2a0addac57}, SpecialFunc None
   Folder Sub: Id {d1926f8b-ff58-44d9-9156-ec5f00475888}
   Method M_AlarmHistory: Id {0e3c3bf5-2da2-4ed3-b7d8-cece9b20ffa6}
   Method M_GetFileName: Id {4c99bb74-f9a5-4074-bb13-078c9bcf604a}
   Method M_ProductionHistory: Id {b278d4fc-53ca-480a-8fab-10f1b6bf22e8}
   Method M_ProductionReport: Id {42b7cd43-4f12-4416-9ca6-76406e00b394}
   Method M_ProductionSummary: Id {0eb07201-11b4-469c-9445-2612e27f826c}
   Method M_RegularCheckResults: Id {4f391bd5-d0aa-4909-93cc-5379d69be5a3}
   Method M_SoDuration: Id {34847b3f-fcce-4d1d-ab8f-2e050ac3309f}
   Method M_StopCount: Id {a1505196-e5cb-459d-bc10-3909af20d9b6} *)
